{attribute 'GeneratedUsingTerminal: EK1122-0000-0018'}
{attribute addProperty BoxType "EK1122-0000-0018"}
{attribute addProperty Id "Beckhoff_EL31xxsub_EK1100EK1100_AB5A94672"}
{attribute addProperty CRC "4127309750"}
{attribute addProperty Size "2"}
TYPE Beckhoff_EL31xxEK1122_F601BFB6 EXTENDS EK1122_AB5A9467 :
STRUCT
	{attribute addProperty Name "Beckhoff_EL31xxsub_EK1100"}
	{attribute addProperty PreviousPort "Beckhoff EL31xxEK1122 : D"}
	Beckhoff_EL31xxsub_EK1100 : EK1100_AB5A9467;
END_STRUCT
END_TYPE

(* stored: Version 1.2.0.0, ProductVersion 3.1.4024.9
   DUT Beckhoff_EL31xxEK1122_F601BFB6: Id {e7b631cb-3561-48bd-99cd-aa6689231588} *)
